// TwinCAT 3 PLC project MC2_PLC
// ProgramVersion: 3.1.4024.0
// libraries:
//   Tc2_MC2, * (Beckhoff Automation GmbH)
//   Tc2_Standard, * (Beckhoff Automation GmbH)
//   Tc2_System, * (Beckhoff Automation GmbH)
//   Tc3_Module, * (Beckhoff Automation GmbH)
// project tree:
//   GVLs/ GVL.TcGVL
//   / PlcTask.TcTTO
//   POUs/ MAIN.TcPOU
// real-time tasks:
//   TASK PlcTask: cycle T#10ms, priority 20, ADS port 350
// motion (NC):
//   TASK NC-Task 1 SAF: cycle T#2ms, priority 4, ADS port 501
//   TASK NC-Task 1 SVB: cycle T#10ms, priority 8, ADS port 511
//   AXIS Axis 1 (id 1)
//     OtherSettings: AllowMotionCmdToSlave=true
//     encoder EncType=1
//     drive DrvType=5
//       Analog: TorqueSetpointScale=10, ScaleFactorActTorque=0.1
//       TimeComp: TaskDelayCycles=1
//     controller CtrType=1
//       CtrPara: PriorControlFactor=1
//         Observer: BandWidth=20
//   AXIS Axis 2 (id 2)
//     OtherSettings: AllowMotionCmdToSlave=true
//     encoder EncType=1
//     drive DrvType=5
//       Analog: TorqueSetpointScale=10, ScaleFactorActTorque=0.1
//       TimeComp: TaskDelayCycles=1
//     controller CtrType=1
//       CtrPara: PriorControlFactor=1
//         Observer: BandWidth=20
// variable links:
//   MC2-PLC Instance <-> NC-Task 1 SAF/Axes/Axis 1
//     PlcTask Inputs/GVL.Axis1.NcToPlc <-> Outputs/ToPlc
//     PlcTask Outputs/GVL.Axis1.PlcToNc <-> Inputs/FromPlc
//   MC2-PLC Instance <-> NC-Task 1 SAF/Axes/Axis 2
//     PlcTask Inputs/GVL.Axis2.NcToPlc <-> Outputs/ToPlc
//     PlcTask Outputs/GVL.Axis2.PlcToNc <-> Inputs/FromPlc

CONFIGURATION MC2_PLC
    RESOURCE PLC ON TwinCAT3
        TASK PlcTask(INTERVAL := T#10ms, PRIORITY := 20);
        PROGRAM MAIN WITH PlcTask : MAIN;
    END_RESOURCE
END_CONFIGURATION

// ---- GVLs/GVL.TcGVL
{attribute 'qualified_only'}
VAR_GLOBAL
	Axis1 : AXIS_REF;
	Axis2 : AXIS_REF;
END_VAR

// ---- POUs/MAIN.TcPOU
PROGRAM MAIN
VAR
	fbMC_Power1: MC_Power;
	xEnable: BOOL;
	xControlPower: BOOL;
	fbMC_Power2: MC_Power;
	lrAxis2_Override: LREAL;
	fmMC_Reset1: MC_Reset;
	xAxisReset: BOOL;
	fmMC_Reset2: MC_Reset
;
	Axis: INT;
	Execute: INT;
	xMachineReset: BOOL;
	fbMC_MoveRelative1: MC_MoveRelative;
	xExecuteDistance: BOOL;
	lrDistance: LREAL;
END_VAR

GVL.Axis1.ReadStatus();
GVL.Axis2.ReadStatus();

IF xControlPower THEN
	xEnable := TRUE;
ELSE
	xEnable := FALSE;
END_IF
fbMC_Power1(
		Axis:= GVL.Axis1, 
		Enable:= xEnable, 
		Enable_Positive:= xEnable, 
		Enable_Negative:= xEnable, 
		Override:= 100.0 
		);
		
fbMC_Power2(
	Axis:= GVL.Axis2, 
	Enable:= xEnable, 
	Enable_Positive:= xEnable, 
	Enable_Negative:= xEnable, 
	Override:= lrAxis2_Override 
	);
	
	IF xMachineReset THEN
		xAxisReset := TRUE;
	ELSE 
		xAxisReset := FALSE;
	END_IF
	
fbMC_MoveRelative1(
	Axis:= GVL.Axis1, 
	Execute:= xExecuteDistance, 
	Distance:= lrDistance, 
	Velocity:= 5.0 
 );
	
	fmMC_Reset1(
		Axis:= GVL.Axis1, 
		Execute:= xAxisReset AND GVL.Axis1.Status.Error
		);
	fmMC_Reset2(
		Axis:= GVL.Axis2, 
		Execute:= xAxisReset AND GVL.Axis2.Status.Error
		);

END_PROGRAM
